FUNCTION_BLOCK AngularAxis EXTENDS SM_AngularAxis;
VAR_INPUT
END_VAR
VAR_OUTPUT
END_VAR
VAR
    _testVar : BOOL;
END_VAR

SUPER^();

END_FUNCTION_BLOCK

(* stored: Version 1.1.0.1, ProductVersion 3.1.4018.5
   POU AngularAxis: Id {7cef5983-5996-4c32-8069-f3adb11c518d}, SpecialFunc None *)
